FUNCTION_BLOCK GreenMasterAI EXTENDS GreenMasterAI_Base
VAR_INPUT
END_VAR
VAR_OUTPUT
END_VAR
VAR
	IO_AI_01: TemperatureInput;
	IO_AI_02: TemperatureInput;
	IO_AI_03: TemperatureInput;
	IO_AI_04: TemperatureInput;
	IO_AI_05: TemperatureInput;
	IO_AI_06: TemperatureInput;
	IO_AI_07: TemperatureInput;
	IO_AI_08: TemperatureInput;
END_VAR


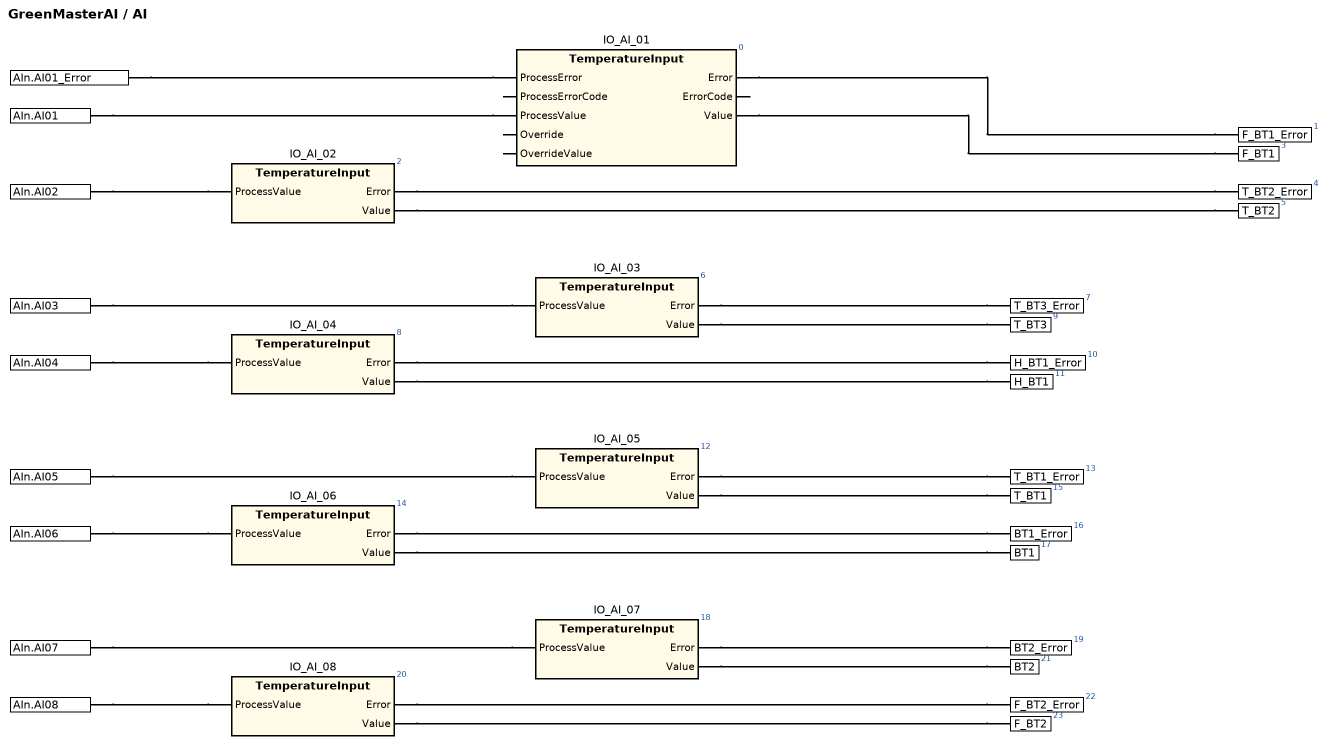
// PAGE AI
IO_AI_01(ProcessError := AIn.AI01_Error, ProcessValue := AIn.AI01); // TemperatureInput
F_BT1_Error := IO_AI_01.Error;
IO_AI_02(ProcessValue := AIn.AI02); // TemperatureInput
F_BT1 := IO_AI_01.Value;
T_BT2_Error := IO_AI_02.Error;
T_BT2 := IO_AI_02.Value;
IO_AI_03(ProcessValue := AIn.AI03); // TemperatureInput
T_BT3_Error := IO_AI_03.Error;
IO_AI_04(ProcessValue := AIn.AI04); // TemperatureInput
T_BT3 := IO_AI_03.Value;
H_BT1_Error := IO_AI_04.Error;
H_BT1 := IO_AI_04.Value;
IO_AI_05(ProcessValue := AIn.AI05); // TemperatureInput
T_BT1_Error := IO_AI_05.Error;
IO_AI_06(ProcessValue := AIn.AI06); // TemperatureInput
T_BT1 := IO_AI_05.Value;
BT1_Error := IO_AI_06.Error;
BT1 := IO_AI_06.Value;
IO_AI_07(ProcessValue := AIn.AI07); // TemperatureInput
BT2_Error := IO_AI_07.Error;
IO_AI_08(ProcessValue := AIn.AI08); // TemperatureInput
BT2 := IO_AI_07.Value;
F_BT2_Error := IO_AI_08.Error;
F_BT2 := IO_AI_08.Value;

END_FUNCTION_BLOCK

(* stored: Version 1.1.0.1, ProductVersion 3.1.4024.4
   POU GreenMasterAI: Id {4d6356ab-9fd2-4c06-baba-c4ef9e296693}, SpecialFunc None *)
